(* CODESYS project IndraLogic.project

Project tree, tasks and I/O mapping:
  IndraMotionMlc1 : IndraControl XM2, Bosch Rexroth AG, order no. dependent on customer specific configuration, version 14.22.36.0
    application Application
      libraries: Linked List, 1.2.1.14 (Bosch Rexroth); MQTT Client, 2.3.8.14 (Bosch Rexroth)
      task PlcTask (cyclic, interval 10 ms, priority 5, watchdog 10 ms x 2) calls PlcProg
      function CheckBounds [ST]
      global variables UserVarGlobal
      Symbols
      program PlcProg [ST]
    S20_I_O : S20_I_O, Bosch Rexroth AG, version 14.22.10.1
      S20_RS_UNI : S20-RS-UNI, Bosch Rexroth AG, order no. R911173343, version Revision=16#0
          settings: Complex Protocol.IDN = 16#010005E3; Complex Protocol.IDN = 16#010005E3; PropritaryParameterSet_P-1-0128.0.0.IDN = 16#01009080; PropritaryParameterSet_P-1-0020.0.0.IDN = 16#01009014; PropritaryParameterSet_P-1-0022.0.0.IDN = 16#01009016
          unmapped channels: S20-RS-UNI - Control, Complex Protocol, S20-RS-UNI - Status, Complex Protocol
    Sercos_III_Master : SercosIII Master, Rexroth, order no. 1, version 14.6.0.0
*)

// IndraMotionMlc1/Application/UserVarGlobal
{attribute 'qualified_only'}
VAR_GLOBAL
END_VAR

// IndraMotionMlc1/Application/PlcProg
PROGRAM PlcProg
VAR
	mqttClient : MQTTClientFB;
	mqttStatusPublish : MQTTPublishFB;
    sStatus : STRING:='ONLINE';
	mqttSubscribe : MQTTSubscribeFB;
	mqttString : MQTTGetStringFB;
	sStatusPC : STRING;
	
END_VAR

mqttClient(
	Enable:= TRUE, 
	IPAddress:= '192.168.99.216' , 
	Port:= 1883, 
	ConnectionTimeout:= , 
	KeepAlive:= 10 , 
	ClientID:= 'plcClient' , 
	Username:= , 
	Password:= , 
	LastWillRetain:= TRUE , 
	LastWillTopic:= 'ORZEL_PLC/STATUS/CONNECTION' , 
	LastWillMessage:= 'OFFLINE' , 
	LastWillQos:=  , 
	TCPConnected=> , 
	Connected=> , 
	Socket=> , 
	PubAckID=> , 
	ErrorCode=> , 
	ErrorInfo=> , 
	ConnectionState=> , 
	SubscribedDataRecvd=> ); 
	


mqttStatusPublish(
	Enable:= TRUE , 
	Post:= , 
	Retained:= TRUE , 
	QoS:= , 
	Topic:='ORZEL_PLC/STATUS/CONNECTION' , 
	Payload:= ADR(sStatus) , 
	DataLength:= INT_TO_UINT(len(sStatus)) , 
	ConnectionHandle:= ADR(mqttClient) , 
	ErrorCode=> , 
	RunningState=> );

mqttSubscribe(
	Enable:= TRUE, 
	Post:= , 
	Topic:= 'ORZEL_PC/STATUS/CONNECTION', 
	QoS:= , 
	ConnectionHandle:= ADR(mqttClient), 
	ErrorCode=> , 
	RunningState=> , 
	Complete=> , 
	Retries=> );

mqttString(
	Enable:= mqttSubscribe.Complete, 
	Topic:= 'ORZEL_PC/STATUS/CONNECTION', 
	Prefix:= , 
	Enabled=> , 
	Output=> sStatusPC, 
	Done=> );
	
IF mqttClient.Connected THEN
	mqttStatusPublish.Post := TRUE;
	mqttSubscribe.Post := TRUE;
ELSE
	mqttStatusPublish.Post := FALSE;
	mqttSubscribe.Post := FALSE;
END_IF

END_PROGRAM

// IndraMotionMlc1/Application/CheckBounds
(*
General Header
----------------------------------------------------------------------------------------------
Short description      : Function to check access to array within valid bounds.
                         After inserting/removing this function, no online-change will be possible! A complete download will be necessary!
Version                : 14.1.0.0
Author                 : DC-IA/EAM3 (MD)
Date                   : 2015-01-12
Company                : Bosch Rexroth AG
Target                 : IndraLogic XLC/MLC
Functional description : This function will be called implicitly before the read/write access
                         to arrays takes places.
                         The index of the subsequent array accesses is checked for valid
                         limits.
                         In case of invalid access, an error is entered in the diagnostic
                         logbook and the application is stopped due to an access violation to
                         avoid machine damage.
                         In this case, check the callstack (menu Debug/Callstack) and modify
                         the faulty logic. 
Handling specials      : This function increases the cycle time of all IEC-tasks using array
                         accesses. 
                         The increase depends on the number of the read/write accesses to
                         arrays.
                         After inserting/removing this function, no online-change will be possible! 
                         A complete download will be necessary!
						 This is an exemplary implementation of the function. 
                         The implementation has to be adjusted to your application/machine.
						 Per default, the PLC-Task will generate an access violation which leads to
                         an application stop and a F5-error with error reaction respectively.
                         Please verify whether this default behaviour can damage your machine 
                         or lead to a complex recommissioning. 
                         In this case, adapt the error reaction to your application.
						 
                         If your application isn't too time-critical, you should leave this function 
						 while commissioning the machine and production in your application.  
                         If you remove this funciton, ensure that your code is faultless.
                         
                         Do not modify the declaration of this function! 
                         Do not change the attributes above the function header!
----------------------------------------------------------------------------------------------
*)
{attribute 'check_bounds'}
{attribute 'no_check'}
{attribute 'signature_flag' := '1073741824'}
FUNCTION CheckBounds : DINT
VAR_INPUT
	index, lower, upper: DINT;
END_VAR
VAR
	{attribute 'hide'}
	bByte: BYTE;
	ptNull: POINTER TO BYTE :=0;
	errstr: STRING;
	
END_VAR

(*************************************************************
This function was generated by the 'check array access'
option of the controllers 'properties' dialog box.
If you delete this comment, the 'check array access' option
of the controllers 'properties' dialog box will be removed.
**************************************************************)
    (**************************************************************************************************)
    (* The implementation has to be adjusted to your application/machine.                             *)
    (* This is an exemplary implementation of the function.                                           *)
    (* Per default, an access violation is generated to avoid machine damage                          *)
    (* Check the Call Stack (menu Debug/Callstack) and modify the faulty logic!                       *)
    (**************************************************************************************************)

IF  index < lower THEN 
	errstr:= 'CheckBounds: Lower arrayindex ';
	errstr:=CONCAT(STR1:=errstr  , STR2:= DINT_TO_STRING(lower));
	errstr:=CONCAT(STR1:=errstr  , STR2:= ' underrunned by ');
	errstr:=CONCAT(STR1:=errstr  , STR2:= DINT_TO_STRING(index));
//  This pragma may be removed: 
	{info 'CheckBounds: Please implement your own error reaction below'}
//  EXAMPLE 1 (default): 
//  Set a F0-Error into the diagnostic- and error memory
//  Triggering an access violation --> Application will be stopped and leads to a F5-Error

  ML_SetDiagEntry(
	Severity:= E_LOG_SEVERITY.ERROR, 
	Class:= E_LOG_CLASS.CLASS_0, 
	Facility:= E_LOG_FACILITY.USER, 
	Code:= 0, 
	Text:= ADR(errstr));

	bByte:=ptNull^;(*triggering an access violation *)

// EXAMPLE 2:
// Limit the faulty index to the lower index 
//     -> no memory will be overwritten
//     -> Keep PLC-task and motion running
// Set a E0-Warning into the diagnostic- and error memory
// NOTE: There is still an implementation error in your application code!

//  ML_SetDiagEntry(
//	Severity:= E_LOG_SEVERITY.WARNING, 
//	Class:= E_LOG_CLASS.CLASS_0, 
//	Facility:= E_LOG_FACILITY.USER, 
//	Code:= 0, 
//	Text:= ADR(errstr));
// 
//	CheckBounds := lower; //access to the lower index only 
//  return;
	
ELSIF  index > upper THEN
	errstr:= 'CheckBounds: Higher arrayindex ';
	errstr:=CONCAT(STR1:=errstr  , STR2:= DINT_TO_STRING(upper));
	errstr:=CONCAT(STR1:=errstr  , STR2:= ' overrunned by ');
	errstr:=CONCAT(STR1:=errstr  , STR2:= DINT_TO_STRING(index));

//  this pragma may be removed: 
	{info 'CheckBounds: Please implement your own error reaction below'}
//  example 1 (default): 
//  set a F0-Error into the diagnostic- and error memory
//  triggering an access violation --> Application will be stopped and leads to a F5-Error

  ML_SetDiagEntry(
	Severity:= E_LOG_SEVERITY.ERROR, 
	Class:= E_LOG_CLASS.CLASS_0, 
	Facility:= E_LOG_FACILITY.USER, 
	Code:= 0, 
	Text:= ADR(errstr));

	bByte:=ptNull^;(*triggering an access violation *)

//example 2:
// Limit the faulty index to the upper index 
//     -> no memory will be overwritten
//     -> Keep PLC-task and motion running
// Set a E0-Warning into the diagnostic- and error memory
// NOTE: There is still an implementation error in your application code!

//  ML_SetDiagEntry(
//	Severity:= E_LOG_SEVERITY.WARNING, 
//	Class:= E_LOG_CLASS.CLASS_0, 
//	Facility:= E_LOG_FACILITY.USER, 
//	Code:= 0, 
//	Text:= ADR(errstr));
// 
//	CheckBounds := upper; //access to the upper index only 
//  return;

ELSE // access to array is ok  
	CheckBounds := index;
END_IF

END_FUNCTION
